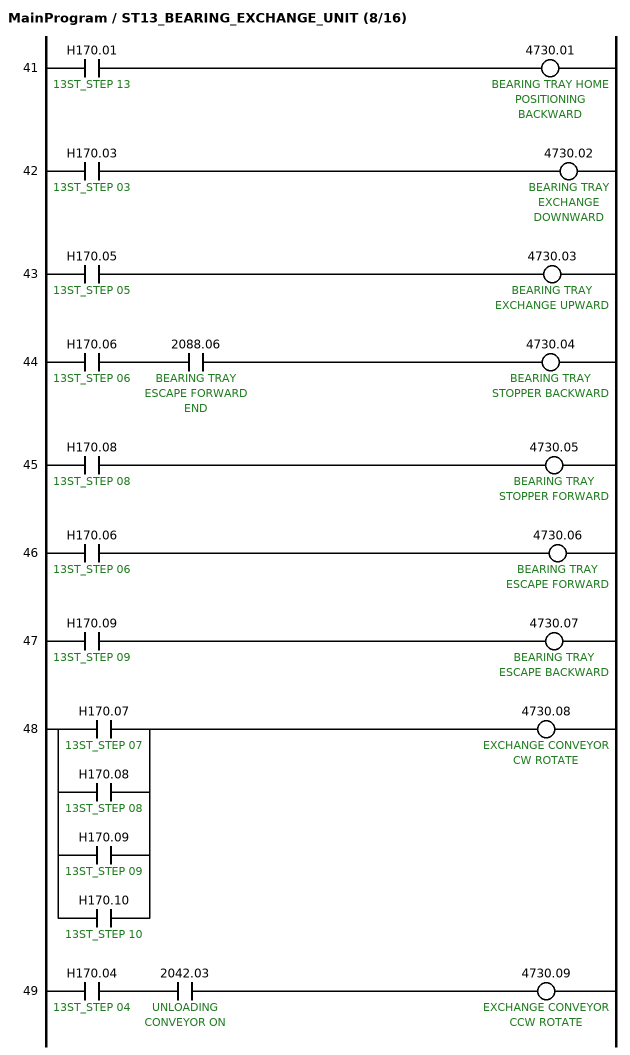
; [picture p600: MainProgram / ST13_BEARING_EXCHANGE_UNIT, rungs 41-49]
; rung 41
LD H170.01  ; 13ST_STEP 13
OUT 4730.01  ; BEARING TRAY HOME POSITIONING BACKWARD
; rung 42
LD H170.03  ; 13ST_STEP 03
OUT 4730.02  ; BEARING TRAY EXCHANGE DOWNWARD
; rung 43
LD H170.05  ; 13ST_STEP 05
OUT 4730.03  ; BEARING TRAY EXCHANGE UPWARD
; rung 44
LD H170.06  ; 13ST_STEP 06
AND 2088.06  ; BEARING TRAY ESCAPE FORWARD END
OUT 4730.04  ; BEARING TRAY STOPPER BACKWARD
; rung 45
LD H170.08  ; 13ST_STEP 08
OUT 4730.05  ; BEARING TRAY STOPPER FORWARD
; rung 46
LD H170.06  ; 13ST_STEP 06
OUT 4730.06  ; BEARING TRAY ESCAPE FORWARD
; rung 47
LD H170.09  ; 13ST_STEP 09
OUT 4730.07  ; BEARING TRAY ESCAPE BACKWARD
; rung 48
LD H170.07  ; 13ST_STEP 07
OR H170.08  ; 13ST_STEP 08
OR H170.09  ; 13ST_STEP 09
OR H170.10  ; 13ST_STEP 10
OUT 4730.08  ; EXCHANGE CONVEYOR CW ROTATE
; rung 49
LD H170.04  ; 13ST_STEP 04
AND 2042.03  ; UNLOADING CONVEYOR ON
OUT 4730.09  ; EXCHANGE CONVEYOR CCW ROTATE

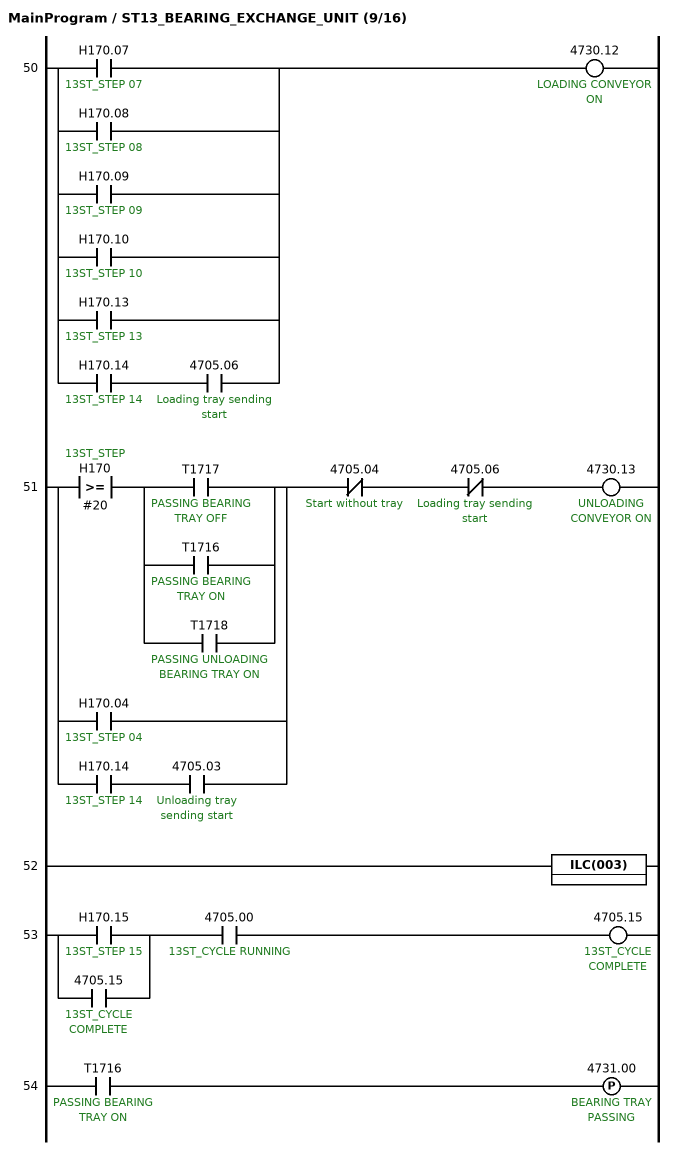
; rung 50
LD H170.07  ; 13ST_STEP 07
OR H170.08  ; 13ST_STEP 08
OR H170.09  ; 13ST_STEP 09
OR H170.10  ; 13ST_STEP 10
OR H170.13  ; 13ST_STEP 13
LD H170.14  ; 13ST_STEP 14
AND 4705.06  ; Loading tray sending start
ORLD
OUT 4730.12  ; LOADING CONVEYOR ON
; rung 51
LD>=(325) H170 #20  ; 13ST_STEP
LD T1717  ; PASSING BEARING TRAY OFF
OR T1716  ; PASSING BEARING TRAY ON
OR T1718  ; PASSING UNLOADING BEARING TRAY ON
ANDLD
OR H170.04  ; 13ST_STEP 04
LD H170.14  ; 13ST_STEP 14
AND 4705.03  ; Unloading tray sending start
ORLD
ANDNOT 4705.04  ; Start without tray
ANDNOT 4705.06  ; Loading tray sending start
OUT 4730.13  ; UNLOADING CONVEYOR ON
; rung 52
ILC(003)
; rung 53
LD H170.15  ; 13ST_STEP 15
OR 4705.15  ; 13ST_CYCLE COMPLETE
AND 4705.00  ; 13ST_CYCLE RUNNING
OUT 4705.15  ; 13ST_CYCLE COMPLETE
; rung 54
LD T1716  ; PASSING BEARING TRAY ON
DIFU(013) 4731.00  ; BEARING TRAY PASSING

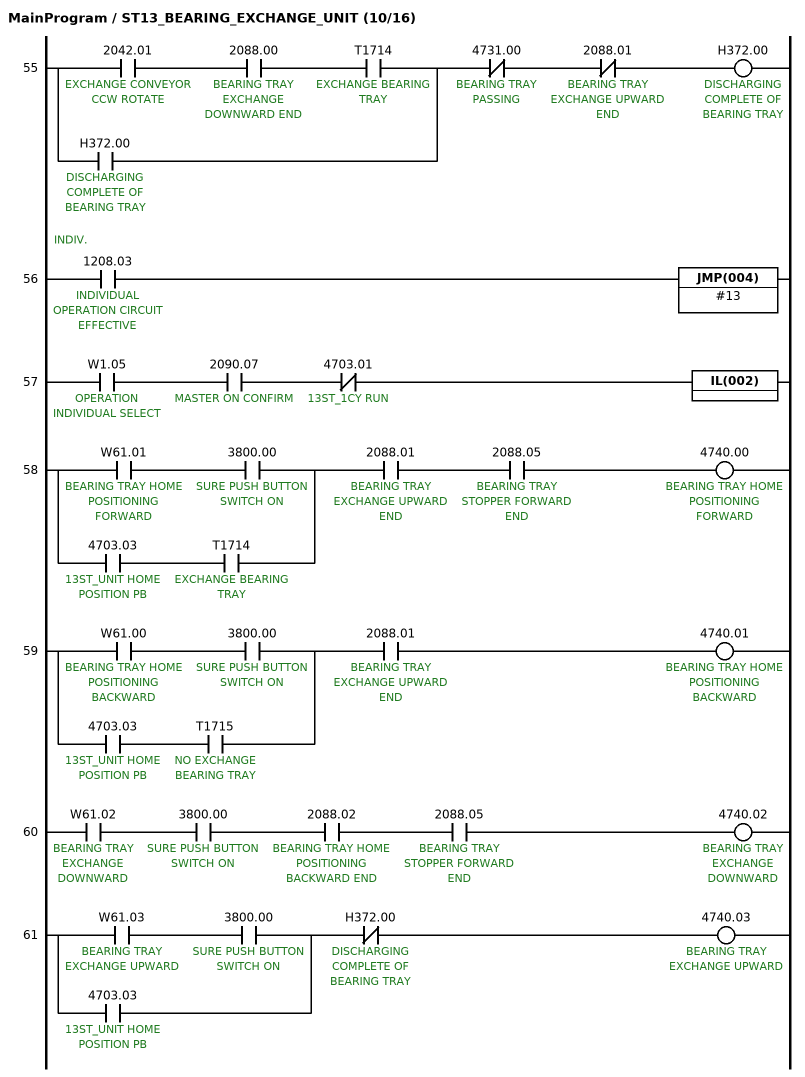
; rung 55
LD 2042.01  ; EXCHANGE CONVEYOR CCW ROTATE
AND 2088.00  ; BEARING TRAY EXCHANGE DOWNWARD END
AND T1714  ; EXCHANGE BEARING TRAY
OR H372.00  ; DISCHARGING COMPLETE OF BEARING TRAY
ANDNOT 4731.00  ; BEARING TRAY PASSING
ANDNOT 2088.01  ; BEARING TRAY EXCHANGE UPWARD END
OUT H372.00  ; DISCHARGING COMPLETE OF BEARING TRAY
; rung 56: INDIV.
LD 1208.03  ; INDIVIDUAL OPERATION CIRCUIT EFFECTIVE
JMP(004) #13
; rung 57
LD W1.05  ; OPERATION INDIVIDUAL SELECT
AND 2090.07  ; MASTER ON CONFIRM
ANDNOT 4703.01  ; 13ST_1CY RUN
IL(002)
; rung 58
LD W61.01  ; BEARING TRAY HOME POSITIONING FORWARD
AND 3800.00  ; SURE PUSH BUTTON SWITCH ON
LD 4703.03  ; 13ST_UNIT HOME POSITION PB
AND T1714  ; EXCHANGE BEARING TRAY
ORLD
AND 2088.01  ; BEARING TRAY EXCHANGE UPWARD END
AND 2088.05  ; BEARING TRAY STOPPER FORWARD END
OUT 4740.00  ; BEARING TRAY HOME POSITIONING FORWARD
; rung 59
LD W61.00  ; BEARING TRAY HOME POSITIONING BACKWARD
AND 3800.00  ; SURE PUSH BUTTON SWITCH ON
LD 4703.03  ; 13ST_UNIT HOME POSITION PB
AND T1715  ; NO EXCHANGE BEARING TRAY
ORLD
AND 2088.01  ; BEARING TRAY EXCHANGE UPWARD END
OUT 4740.01  ; BEARING TRAY HOME POSITIONING BACKWARD
; rung 60
LD W61.02  ; BEARING TRAY EXCHANGE DOWNWARD
AND 3800.00  ; SURE PUSH BUTTON SWITCH ON
AND 2088.02  ; BEARING TRAY HOME POSITIONING BACKWARD END
AND 2088.05  ; BEARING TRAY STOPPER FORWARD END
OUT 4740.02  ; BEARING TRAY EXCHANGE DOWNWARD
; rung 61
LD W61.03  ; BEARING TRAY EXCHANGE UPWARD
AND 3800.00  ; SURE PUSH BUTTON SWITCH ON
OR 4703.03  ; 13ST_UNIT HOME POSITION PB
ANDNOT H372.00  ; DISCHARGING COMPLETE OF BEARING TRAY
OUT 4740.03  ; BEARING TRAY EXCHANGE UPWARD

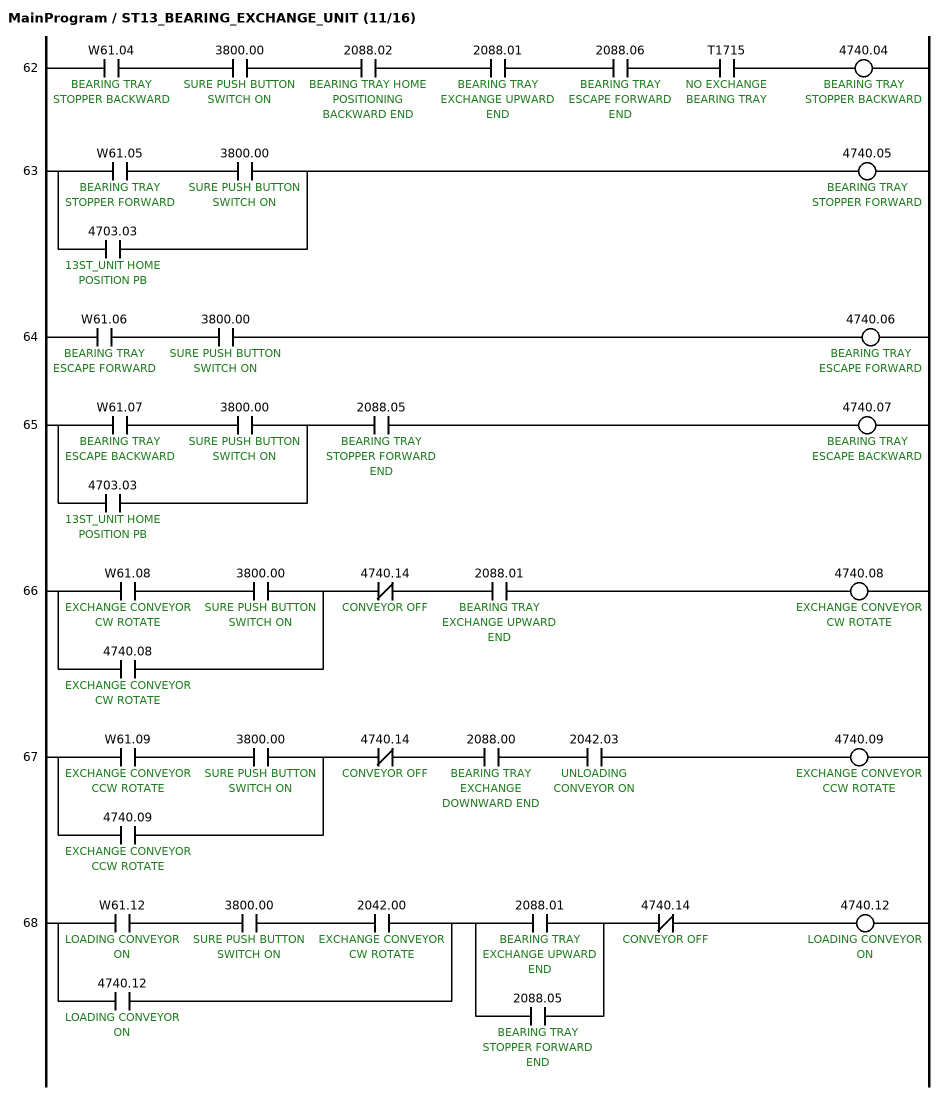
; rung 62
LD W61.04  ; BEARING TRAY STOPPER BACKWARD
AND 3800.00  ; SURE PUSH BUTTON SWITCH ON
AND 2088.02  ; BEARING TRAY HOME POSITIONING BACKWARD END
AND 2088.01  ; BEARING TRAY EXCHANGE UPWARD END
AND 2088.06  ; BEARING TRAY ESCAPE FORWARD END
AND T1715  ; NO EXCHANGE BEARING TRAY
OUT 4740.04  ; BEARING TRAY STOPPER BACKWARD
; rung 63
LD W61.05  ; BEARING TRAY STOPPER FORWARD
AND 3800.00  ; SURE PUSH BUTTON SWITCH ON
OR 4703.03  ; 13ST_UNIT HOME POSITION PB
OUT 4740.05  ; BEARING TRAY STOPPER FORWARD
; rung 64
LD W61.06  ; BEARING TRAY ESCAPE FORWARD
AND 3800.00  ; SURE PUSH BUTTON SWITCH ON
OUT 4740.06  ; BEARING TRAY ESCAPE FORWARD
; rung 65
LD W61.07  ; BEARING TRAY ESCAPE BACKWARD
AND 3800.00  ; SURE PUSH BUTTON SWITCH ON
OR 4703.03  ; 13ST_UNIT HOME POSITION PB
AND 2088.05  ; BEARING TRAY STOPPER FORWARD END
OUT 4740.07  ; BEARING TRAY ESCAPE BACKWARD
; rung 66
LD W61.08  ; EXCHANGE CONVEYOR CW ROTATE
AND 3800.00  ; SURE PUSH BUTTON SWITCH ON
OR 4740.08  ; EXCHANGE CONVEYOR CW ROTATE
ANDNOT 4740.14  ; CONVEYOR OFF
AND 2088.01  ; BEARING TRAY EXCHANGE UPWARD END
OUT 4740.08  ; EXCHANGE CONVEYOR CW ROTATE
; rung 67
LD W61.09  ; EXCHANGE CONVEYOR CCW ROTATE
AND 3800.00  ; SURE PUSH BUTTON SWITCH ON
OR 4740.09  ; EXCHANGE CONVEYOR CCW ROTATE
ANDNOT 4740.14  ; CONVEYOR OFF
AND 2088.00  ; BEARING TRAY EXCHANGE DOWNWARD END
AND 2042.03  ; UNLOADING CONVEYOR ON
OUT 4740.09  ; EXCHANGE CONVEYOR CCW ROTATE
; rung 68
LD W61.12  ; LOADING CONVEYOR ON
AND 3800.00  ; SURE PUSH BUTTON SWITCH ON
AND 2042.00  ; EXCHANGE CONVEYOR CW ROTATE
OR 4740.12  ; LOADING CONVEYOR ON
LD 2088.01  ; BEARING TRAY EXCHANGE UPWARD END
OR 2088.05  ; BEARING TRAY STOPPER FORWARD END
ANDLD
ANDNOT 4740.14  ; CONVEYOR OFF
OUT 4740.12  ; LOADING CONVEYOR ON

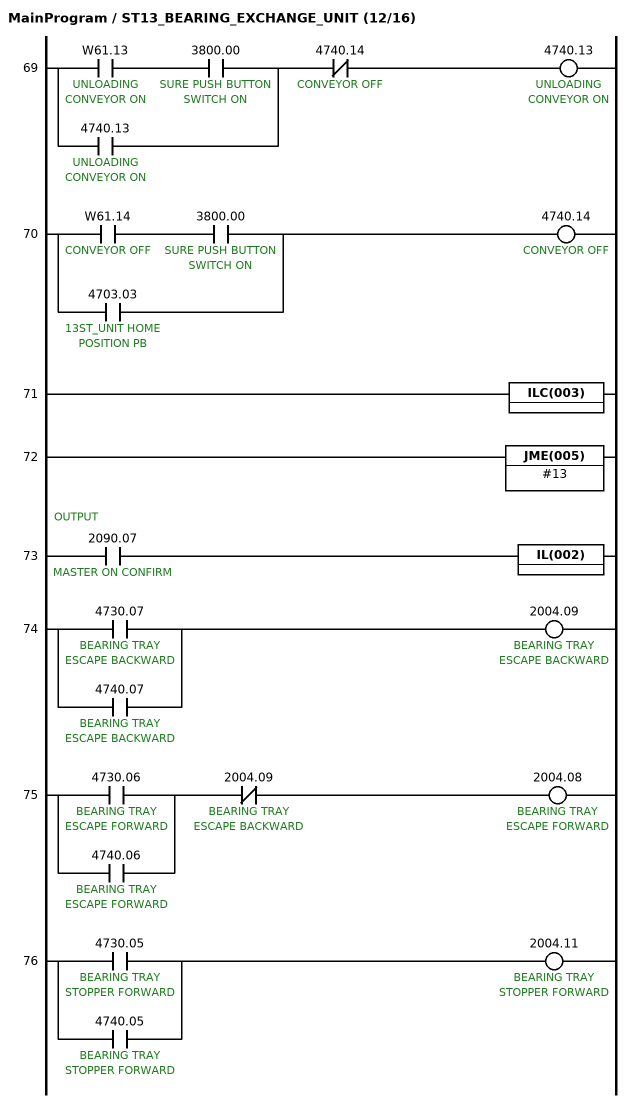
; rung 69
LD W61.13  ; UNLOADING CONVEYOR ON
AND 3800.00  ; SURE PUSH BUTTON SWITCH ON
OR 4740.13  ; UNLOADING CONVEYOR ON
ANDNOT 4740.14  ; CONVEYOR OFF
OUT 4740.13  ; UNLOADING CONVEYOR ON
; rung 70
LD W61.14  ; CONVEYOR OFF
AND 3800.00  ; SURE PUSH BUTTON SWITCH ON
OR 4703.03  ; 13ST_UNIT HOME POSITION PB
OUT 4740.14  ; CONVEYOR OFF
; rung 71
ILC(003)
; rung 72
JME(005) #13
; rung 73: OUTPUT
LD 2090.07  ; MASTER ON CONFIRM
IL(002)
; rung 74
LD 4730.07  ; BEARING TRAY ESCAPE BACKWARD
OR 4740.07  ; BEARING TRAY ESCAPE BACKWARD
OUT 2004.09  ; BEARING TRAY ESCAPE BACKWARD
; rung 75
LD 4730.06  ; BEARING TRAY ESCAPE FORWARD
OR 4740.06  ; BEARING TRAY ESCAPE FORWARD
ANDNOT 2004.09  ; BEARING TRAY ESCAPE BACKWARD
OUT 2004.08  ; BEARING TRAY ESCAPE FORWARD
; rung 76
LD 4730.05  ; BEARING TRAY STOPPER FORWARD
OR 4740.05  ; BEARING TRAY STOPPER FORWARD
OUT 2004.11  ; BEARING TRAY STOPPER FORWARD

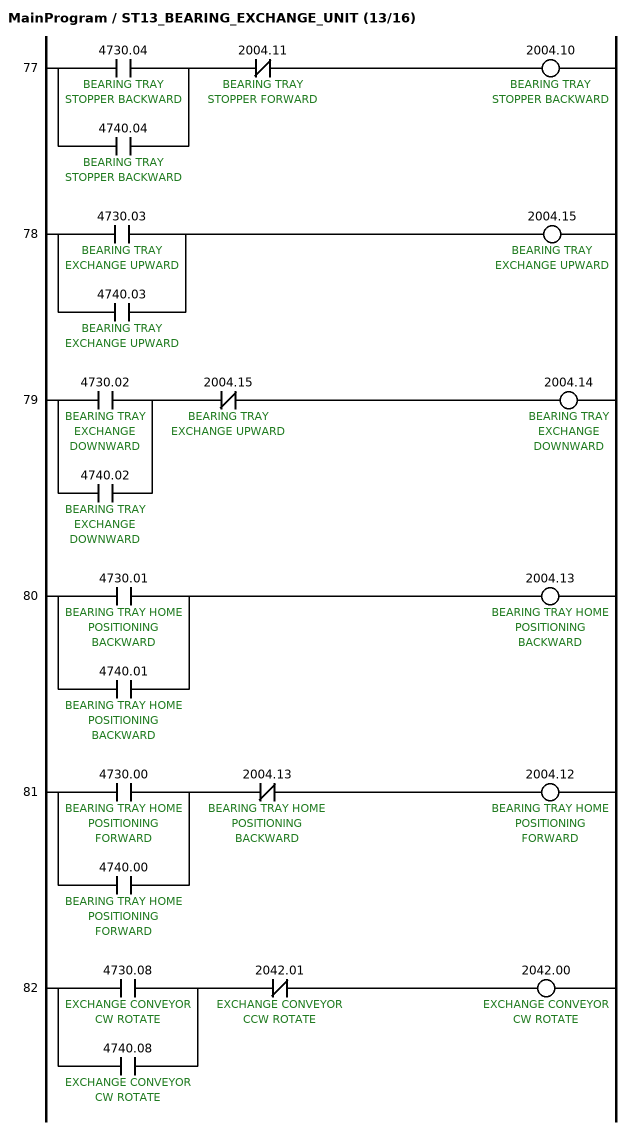
; rung 77
LD 4730.04  ; BEARING TRAY STOPPER BACKWARD
OR 4740.04  ; BEARING TRAY STOPPER BACKWARD
ANDNOT 2004.11  ; BEARING TRAY STOPPER FORWARD
OUT 2004.10  ; BEARING TRAY STOPPER BACKWARD
; rung 78
LD 4730.03  ; BEARING TRAY EXCHANGE UPWARD
OR 4740.03  ; BEARING TRAY EXCHANGE UPWARD
OUT 2004.15  ; BEARING TRAY EXCHANGE UPWARD
; rung 79
LD 4730.02  ; BEARING TRAY EXCHANGE DOWNWARD
OR 4740.02  ; BEARING TRAY EXCHANGE DOWNWARD
ANDNOT 2004.15  ; BEARING TRAY EXCHANGE UPWARD
OUT 2004.14  ; BEARING TRAY EXCHANGE DOWNWARD
; rung 80
LD 4730.01  ; BEARING TRAY HOME POSITIONING BACKWARD
OR 4740.01  ; BEARING TRAY HOME POSITIONING BACKWARD
OUT 2004.13  ; BEARING TRAY HOME POSITIONING BACKWARD
; rung 81
LD 4730.00  ; BEARING TRAY HOME POSITIONING FORWARD
OR 4740.00  ; BEARING TRAY HOME POSITIONING FORWARD
ANDNOT 2004.13  ; BEARING TRAY HOME POSITIONING BACKWARD
OUT 2004.12  ; BEARING TRAY HOME POSITIONING FORWARD
; rung 82
LD 4730.08  ; EXCHANGE CONVEYOR CW ROTATE
OR 4740.08  ; EXCHANGE CONVEYOR CW ROTATE
ANDNOT 2042.01  ; EXCHANGE CONVEYOR CCW ROTATE
OUT 2042.00  ; EXCHANGE CONVEYOR CW ROTATE

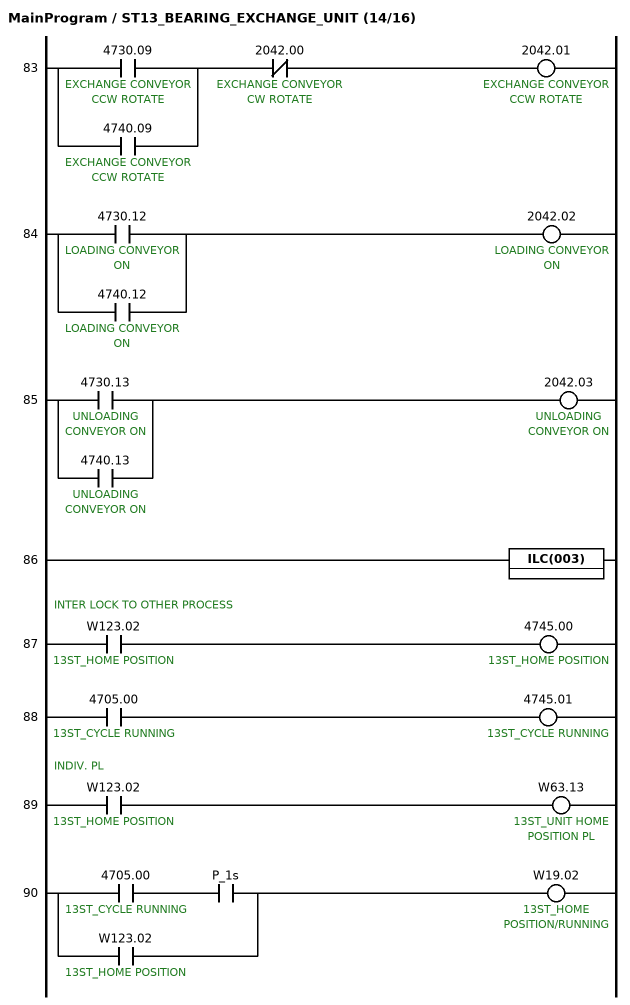
; rung 83
LD 4730.09  ; EXCHANGE CONVEYOR CCW ROTATE
OR 4740.09  ; EXCHANGE CONVEYOR CCW ROTATE
ANDNOT 2042.00  ; EXCHANGE CONVEYOR CW ROTATE
OUT 2042.01  ; EXCHANGE CONVEYOR CCW ROTATE
; rung 84
LD 4730.12  ; LOADING CONVEYOR ON
OR 4740.12  ; LOADING CONVEYOR ON
OUT 2042.02  ; LOADING CONVEYOR ON
; rung 85
LD 4730.13  ; UNLOADING CONVEYOR ON
OR 4740.13  ; UNLOADING CONVEYOR ON
OUT 2042.03  ; UNLOADING CONVEYOR ON
; rung 86
ILC(003)
; rung 87: INTER LOCK TO OTHER PROCESS
LD W123.02  ; 13ST_HOME POSITION
OUT 4745.00  ; 13ST_HOME POSITION
; rung 88
LD 4705.00  ; 13ST_CYCLE RUNNING
OUT 4745.01  ; 13ST_CYCLE RUNNING
; rung 89: INDIV. PL
LD W123.02  ; 13ST_HOME POSITION
OUT W63.13  ; 13ST_UNIT HOME POSITION PL
; rung 90
LD 4705.00  ; 13ST_CYCLE RUNNING
AND P_1s
OR W123.02  ; 13ST_HOME POSITION
OUT W19.02  ; 13ST_HOME POSITION/RUNNING

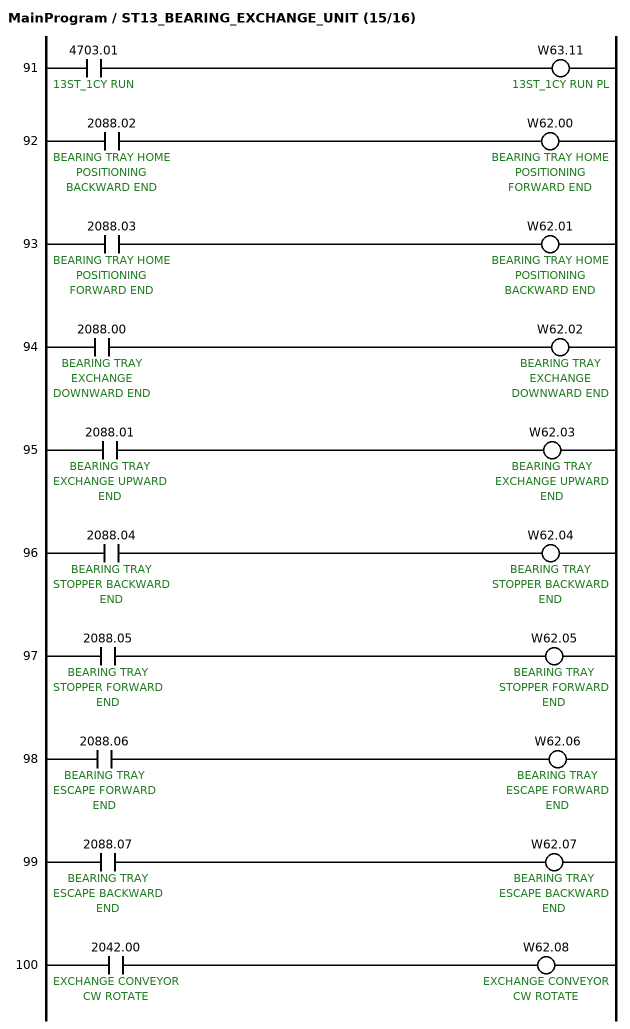
; rung 91
LD 4703.01  ; 13ST_1CY RUN
OUT W63.11  ; 13ST_1CY RUN PL
; rung 92
LD 2088.02  ; BEARING TRAY HOME POSITIONING BACKWARD END
OUT W62.00  ; BEARING TRAY HOME POSITIONING FORWARD END
; rung 93
LD 2088.03  ; BEARING TRAY HOME POSITIONING FORWARD END
OUT W62.01  ; BEARING TRAY HOME POSITIONING BACKWARD END
; rung 94
LD 2088.00  ; BEARING TRAY EXCHANGE DOWNWARD END
OUT W62.02  ; BEARING TRAY EXCHANGE DOWNWARD END
; rung 95
LD 2088.01  ; BEARING TRAY EXCHANGE UPWARD END
OUT W62.03  ; BEARING TRAY EXCHANGE UPWARD END
; rung 96
LD 2088.04  ; BEARING TRAY STOPPER BACKWARD END
OUT W62.04  ; BEARING TRAY STOPPER BACKWARD END
; rung 97
LD 2088.05  ; BEARING TRAY STOPPER FORWARD END
OUT W62.05  ; BEARING TRAY STOPPER FORWARD END
; rung 98
LD 2088.06  ; BEARING TRAY ESCAPE FORWARD END
OUT W62.06  ; BEARING TRAY ESCAPE FORWARD END
; rung 99
LD 2088.07  ; BEARING TRAY ESCAPE BACKWARD END
OUT W62.07  ; BEARING TRAY ESCAPE BACKWARD END
; rung 100
LD 2042.00  ; EXCHANGE CONVEYOR CW ROTATE
OUT W62.08  ; EXCHANGE CONVEYOR CW ROTATE

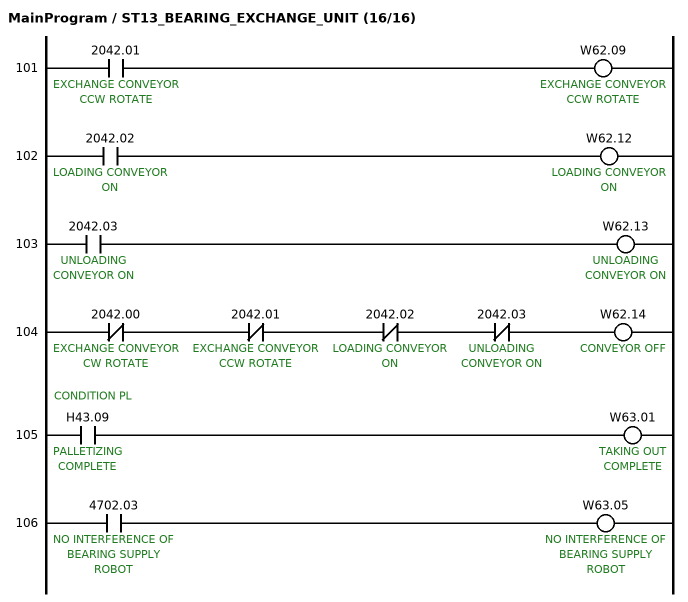
; rung 101
LD 2042.01  ; EXCHANGE CONVEYOR CCW ROTATE
OUT W62.09  ; EXCHANGE CONVEYOR CCW ROTATE
; rung 102
LD 2042.02  ; LOADING CONVEYOR ON
OUT W62.12  ; LOADING CONVEYOR ON
; rung 103
LD 2042.03  ; UNLOADING CONVEYOR ON
OUT W62.13  ; UNLOADING CONVEYOR ON
; rung 104
LDNOT 2042.00  ; EXCHANGE CONVEYOR CW ROTATE
ANDNOT 2042.01  ; EXCHANGE CONVEYOR CCW ROTATE
ANDNOT 2042.02  ; LOADING CONVEYOR ON
ANDNOT 2042.03  ; UNLOADING CONVEYOR ON
OUT W62.14  ; CONVEYOR OFF
; rung 105: CONDITION PL
LD H43.09  ; PALLETIZING COMPLETE
OUT W63.01  ; TAKING OUT COMPLETE
; rung 106
LD 4702.03  ; NO INTERFERENCE OF BEARING SUPPLY ROBOT
OUT W63.05  ; NO INTERFERENCE OF BEARING SUPPLY ROBOT

### Section ST14_DEFECT_DISCHARGE_UNIT
; rung 0: 14ST_DEFECT DISCHARGE UNIT

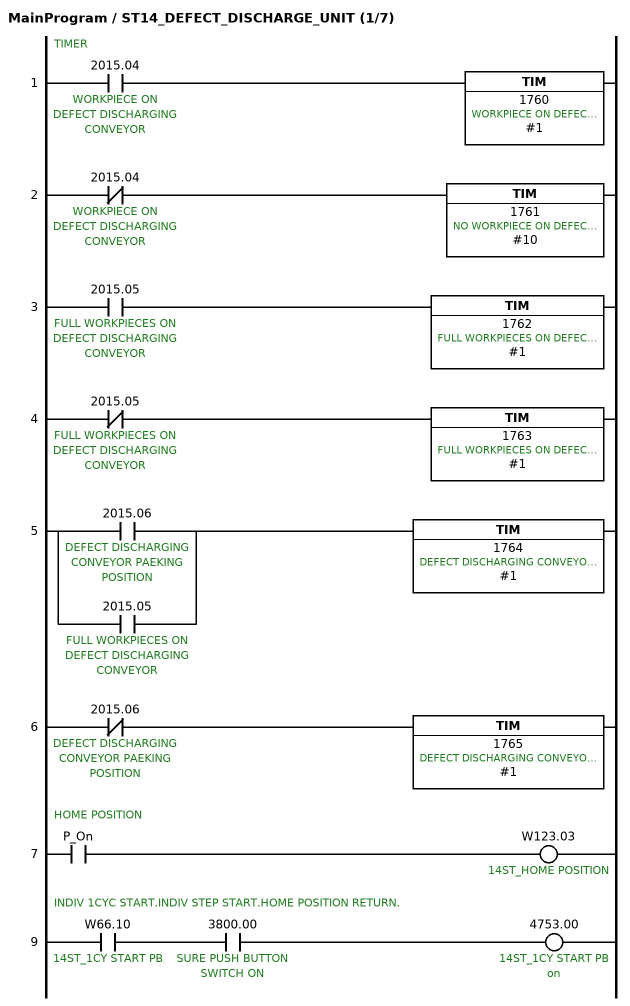
; rung 1: TIMER
LD 2015.04  ; WORKPIECE ON DEFECT DISCHARGING CONVEYOR
TIM 1760 #1  ; WORKPIECE ON DEFECT DISCHARGING CONVEYOR
; rung 2
LDNOT 2015.04  ; WORKPIECE ON DEFECT DISCHARGING CONVEYOR
TIM 1761 #10  ; NO WORKPIECE ON DEFECT DISCHARGING CONVEYOR
; rung 3
LD 2015.05  ; FULL WORKPIECES ON DEFECT DISCHARGING CONVEYOR
TIM 1762 #1  ; FULL WORKPIECES ON DEFECT DISCHARGING CONVEYOR IS TURNED ON
; rung 4
LDNOT 2015.05  ; FULL WORKPIECES ON DEFECT DISCHARGING CONVEYOR
TIM 1763 #1  ; FULL WORKPIECES ON DEFECT DISCHARGING CONVEYOR IS TURNED OFF
; rung 5
LD 2015.06  ; DEFECT DISCHARGING CONVEYOR PAEKING POSITION
OR 2015.05  ; FULL WORKPIECES ON DEFECT DISCHARGING CONVEYOR
TIM 1764 #1  ; DEFECT DISCHARGING CONVEYOR PAEKING POSITION IS TURNED ON
; rung 6
LDNOT 2015.06  ; DEFECT DISCHARGING CONVEYOR PAEKING POSITION
TIM 1765 #1  ; DEFECT DISCHARGING CONVEYOR PAEKING POSITION IS TURNED OFF
; rung 7: HOME POSITION
LD P_On
OUT W123.03  ; 14ST_HOME POSITION
; rung 8: INTERFERENCE
; rung 9: INDIV 1CYC START.INDIV STEP START.HOME POSITION RETURN.
LD W66.10  ; 14ST_1CY START PB
AND 3800.00  ; SURE PUSH BUTTON SWITCH ON
OUT 4753.00  ; 14ST_1CY START PB on

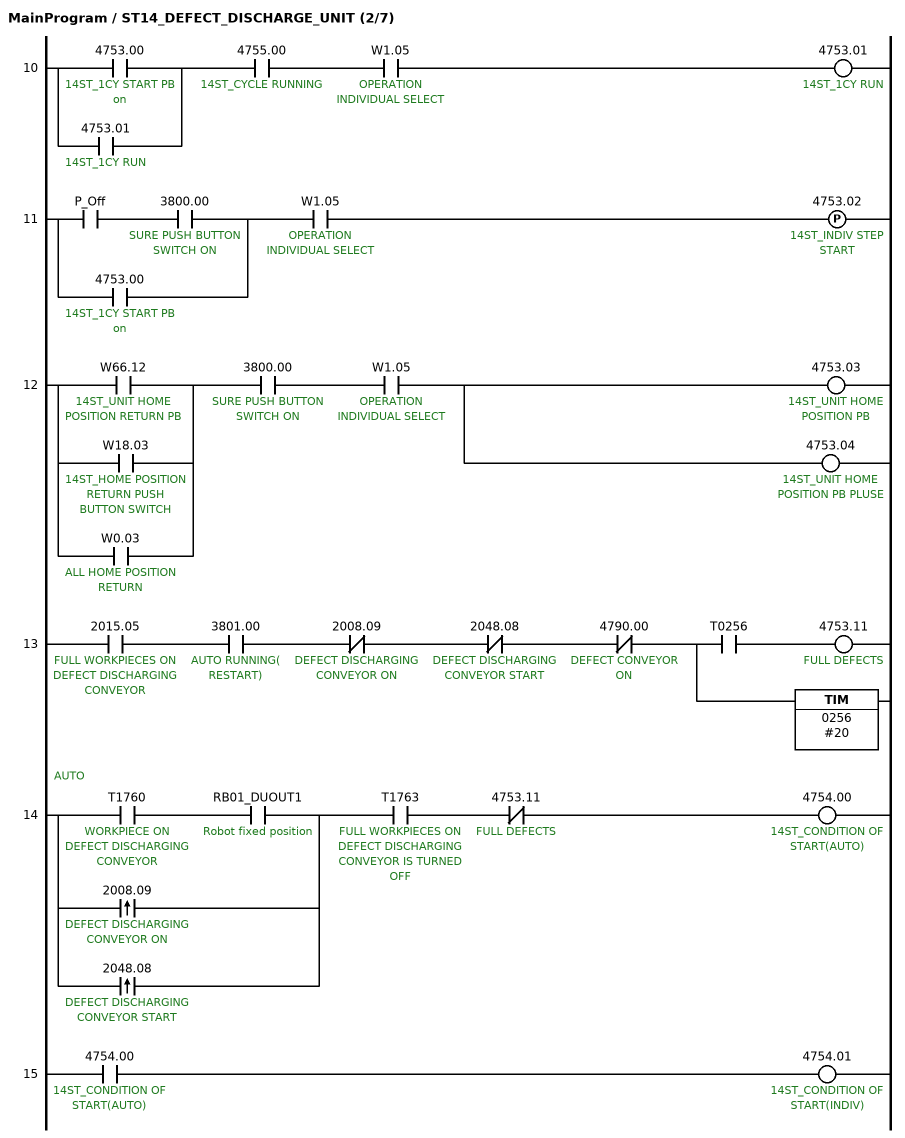
; rung 10
LD 4753.00  ; 14ST_1CY START PB on
OR 4753.01  ; 14ST_1CY RUN
AND 4755.00  ; 14ST_CYCLE RUNNING
AND W1.05  ; OPERATION INDIVIDUAL SELECT
OUT 4753.01  ; 14ST_1CY RUN
; rung 11
LD P_Off
AND 3800.00  ; SURE PUSH BUTTON SWITCH ON
OR 4753.00  ; 14ST_1CY START PB on
AND W1.05  ; OPERATION INDIVIDUAL SELECT
DIFU(013) 4753.02  ; 14ST_INDIV STEP START
; rung 12
LD W66.12  ; 14ST_UNIT HOME POSITION RETURN PB
OR W18.03  ; 14ST_HOME POSITION RETURN PUSH BUTTON SWITCH
OR W0.03  ; ALL HOME POSITION RETURN
AND 3800.00  ; SURE PUSH BUTTON SWITCH ON
AND W1.05  ; OPERATION INDIVIDUAL SELECT
OUT 4753.03  ; 14ST_UNIT HOME POSITION PB
OUT 4753.04  ; 14ST_UNIT HOME POSITION PB PLUSE
; rung 13
LD 2015.05  ; FULL WORKPIECES ON DEFECT DISCHARGING CONVEYOR
AND 3801.00  ; AUTO RUNNING(RESTART)
ANDNOT 2008.09  ; DEFECT DISCHARGING CONVEYOR ON
ANDNOT 2048.08  ; DEFECT DISCHARGING CONVEYOR START
ANDNOT 4790.00  ; DEFECT CONVEYOR ON
OUT TR0
AND T0256
OUT 4753.11  ; FULL DEFECTS
LD TR0
TIM 0256 #20
; rung 14: AUTO
LD T1760  ; WORKPIECE ON DEFECT DISCHARGING CONVEYOR
AND RB01_DUOUT1  ; Robot fixed position
@OR 2008.09  ; DEFECT DISCHARGING CONVEYOR ON
@OR 2048.08  ; DEFECT DISCHARGING CONVEYOR START
AND T1763  ; FULL WORKPIECES ON DEFECT DISCHARGING CONVEYOR IS TURNED OFF
ANDNOT 4753.11  ; FULL DEFECTS
OUT 4754.00  ; 14ST_CONDITION OF START(AUTO)
; rung 15
LD 4754.00  ; 14ST_CONDITION OF START(AUTO)
OUT 4754.01  ; 14ST_CONDITION OF START(INDIV)

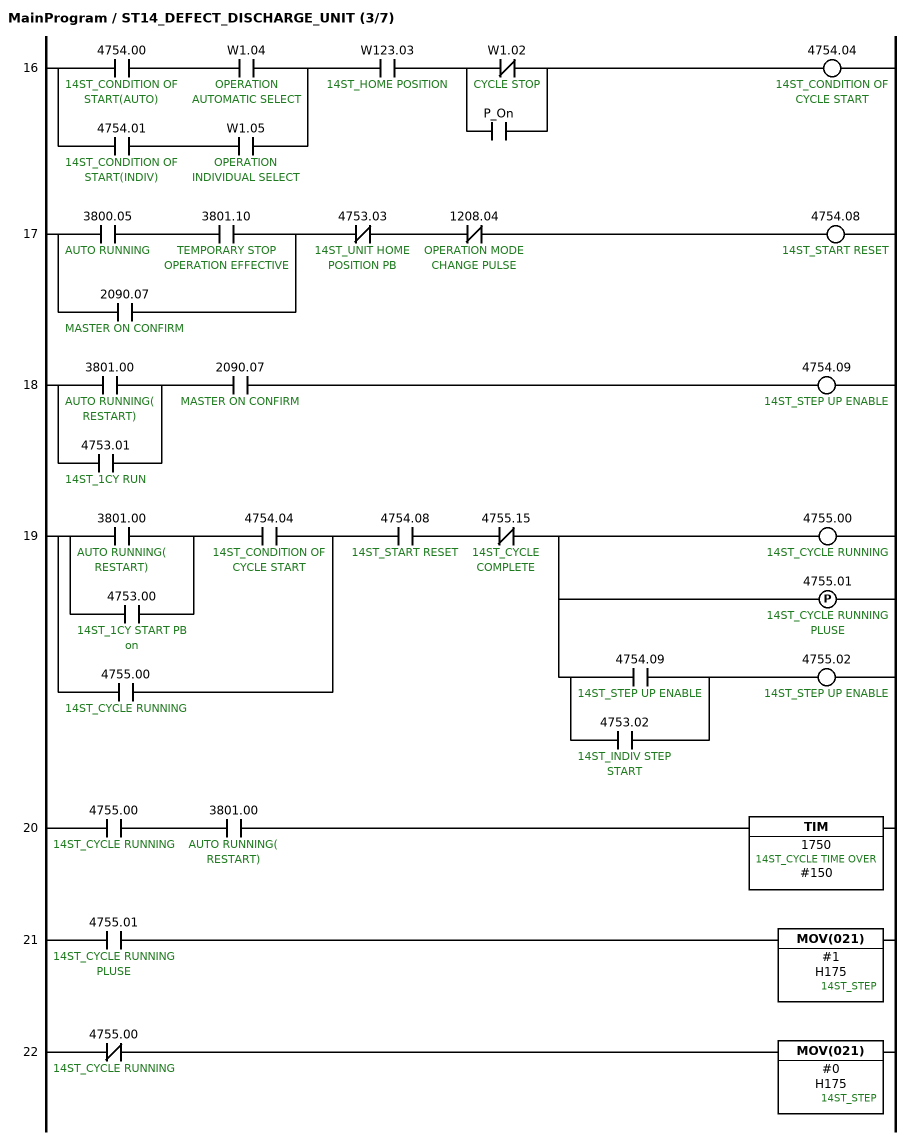
; rung 16
LD 4754.00  ; 14ST_CONDITION OF START(AUTO)
AND W1.04  ; OPERATION AUTOMATIC SELECT
LD 4754.01  ; 14ST_CONDITION OF START(INDIV)
AND W1.05  ; OPERATION INDIVIDUAL SELECT
ORLD
AND W123.03  ; 14ST_HOME POSITION
LDNOT W1.02  ; CYCLE STOP
OR P_On
ANDLD
OUT 4754.04  ; 14ST_CONDITION OF CYCLE START
; rung 17
LD 3800.05  ; AUTO RUNNING
AND 3801.10  ; TEMPORARY STOP OPERATION EFFECTIVE
OR 2090.07  ; MASTER ON CONFIRM
ANDNOT 4753.03  ; 14ST_UNIT HOME POSITION PB
ANDNOT 1208.04  ; OPERATION MODE CHANGE PULSE
OUT 4754.08  ; 14ST_START RESET
; rung 18
LD 3801.00  ; AUTO RUNNING(RESTART)
OR 4753.01  ; 14ST_1CY RUN
AND 2090.07  ; MASTER ON CONFIRM
OUT 4754.09  ; 14ST_STEP UP ENABLE
; rung 19
LD 3801.00  ; AUTO RUNNING(RESTART)
OR 4753.00  ; 14ST_1CY START PB on
AND 4754.04  ; 14ST_CONDITION OF CYCLE START
OR 4755.00  ; 14ST_CYCLE RUNNING
AND 4754.08  ; 14ST_START RESET
ANDNOT 4755.15  ; 14ST_CYCLE COMPLETE
OUT 4755.00  ; 14ST_CYCLE RUNNING
DIFU(013) 4755.01  ; 14ST_CYCLE RUNNING PLUSE
LD 4754.09  ; 14ST_STEP UP ENABLE
OR 4753.02  ; 14ST_INDIV STEP START
ANDLD
OUT 4755.02  ; 14ST_STEP UP ENABLE
; rung 20
LD 4755.00  ; 14ST_CYCLE RUNNING
AND 3801.00  ; AUTO RUNNING(RESTART)
TIM 1750 #150  ; 14ST_CYCLE TIME OVER
; rung 21
LD 4755.01  ; 14ST_CYCLE RUNNING PLUSE
MOV(021) #1 H175  ; 14ST_STEP
; rung 22
LDNOT 4755.00  ; 14ST_CYCLE RUNNING
MOV(021) #0 H175  ; 14ST_STEP

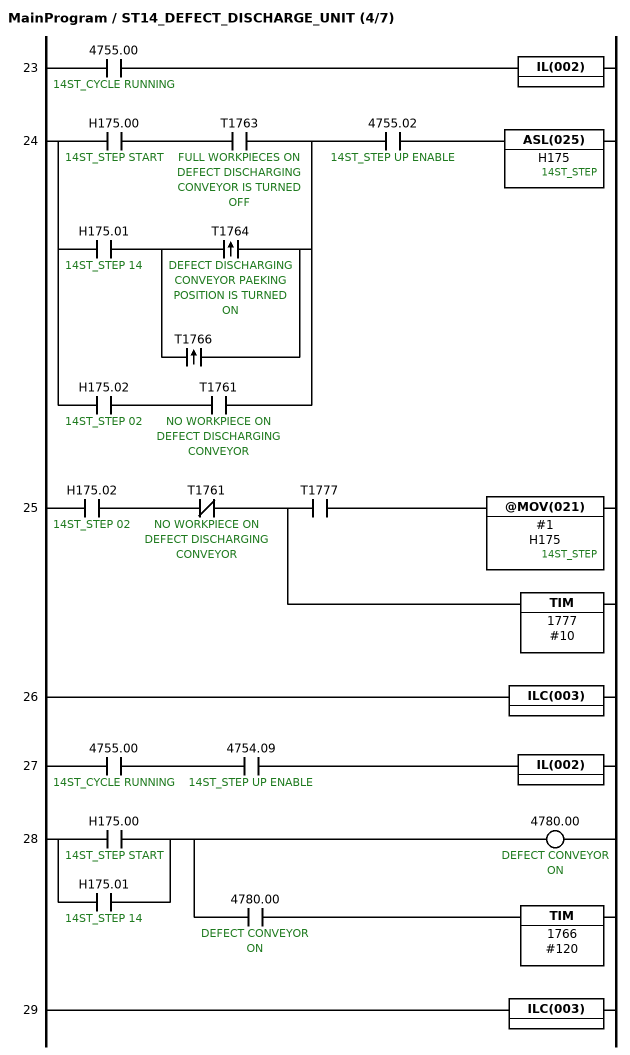
; rung 23
LD 4755.00  ; 14ST_CYCLE RUNNING
IL(002)
; rung 24
LD H175.00  ; 14ST_STEP START
AND T1763  ; FULL WORKPIECES ON DEFECT DISCHARGING CONVEYOR IS TURNED OFF
LD H175.01  ; 14ST_STEP 14
@LD T1764  ; DEFECT DISCHARGING CONVEYOR PAEKING POSITION IS TURNED ON
@OR T1766
ANDLD
ORLD
LD H175.02  ; 14ST_STEP 02
AND T1761  ; NO WORKPIECE ON DEFECT DISCHARGING CONVEYOR
ORLD
AND 4755.02  ; 14ST_STEP UP ENABLE
ASL(025) H175  ; 14ST_STEP
; rung 25
LD H175.02  ; 14ST_STEP 02
ANDNOT T1761  ; NO WORKPIECE ON DEFECT DISCHARGING CONVEYOR
OUT TR0
AND T1777
@MOV(021) #1 H175  ; 14ST_STEP
LD TR0
TIM 1777 #10
; rung 26
ILC(003)
; rung 27
LD 4755.00  ; 14ST_CYCLE RUNNING
AND 4754.09  ; 14ST_STEP UP ENABLE
IL(002)
; rung 28
LD H175.00  ; 14ST_STEP START
OR H175.01  ; 14ST_STEP 14
OUT 4780.00  ; DEFECT CONVEYOR ON
AND 4780.00  ; DEFECT CONVEYOR ON
TIM 1766 #120
; rung 29
ILC(003)

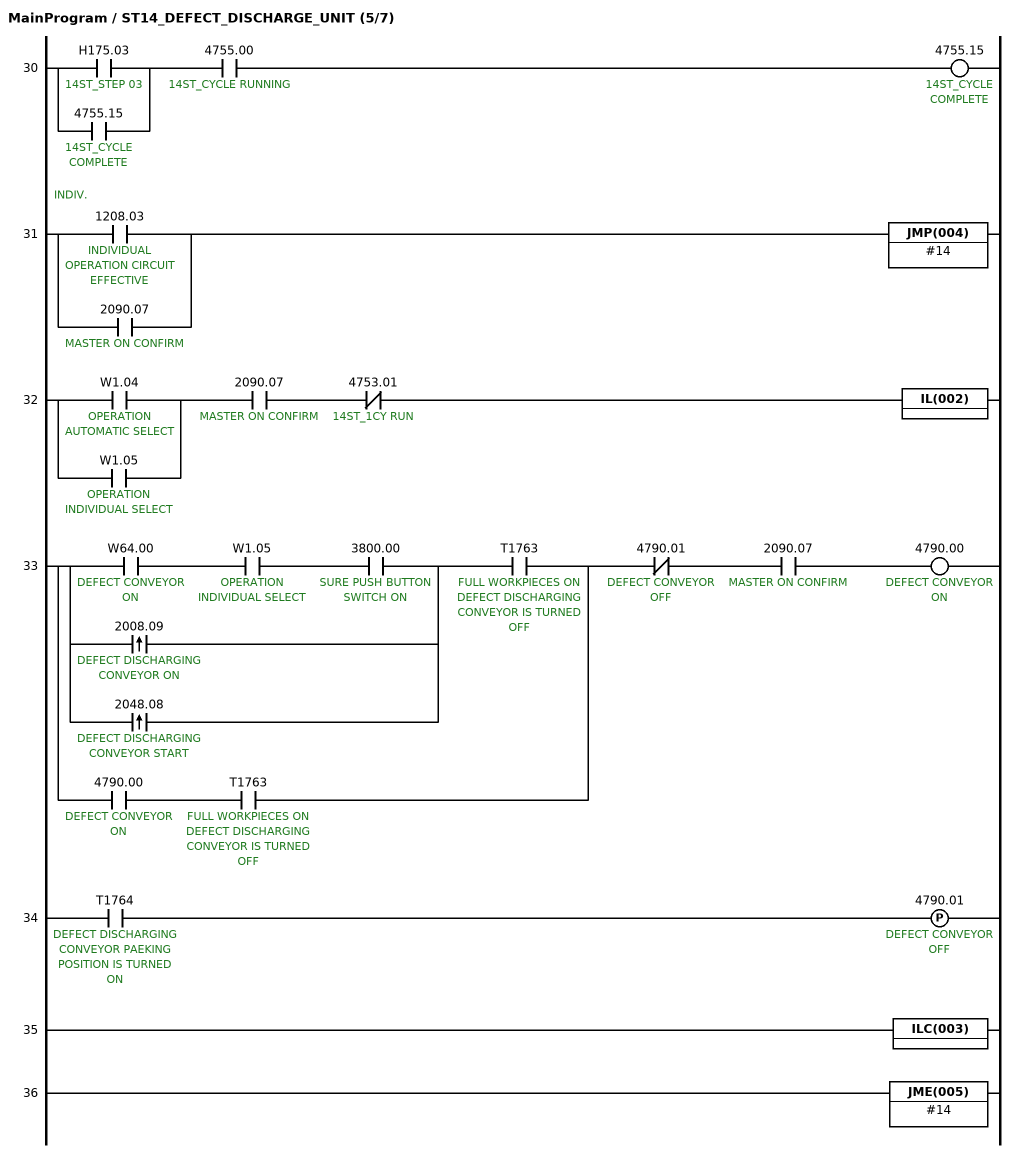
; rung 30
LD H175.03  ; 14ST_STEP 03
OR 4755.15  ; 14ST_CYCLE COMPLETE
AND 4755.00  ; 14ST_CYCLE RUNNING
OUT 4755.15  ; 14ST_CYCLE COMPLETE
; rung 31: INDIV.
LD 1208.03  ; INDIVIDUAL OPERATION CIRCUIT EFFECTIVE
OR 2090.07  ; MASTER ON CONFIRM
JMP(004) #14
; rung 32
LD W1.04  ; OPERATION AUTOMATIC SELECT
OR W1.05  ; OPERATION INDIVIDUAL SELECT
AND 2090.07  ; MASTER ON CONFIRM
ANDNOT 4753.01  ; 14ST_1CY RUN
IL(002)
; rung 33
LD W64.00  ; DEFECT CONVEYOR ON
AND W1.05  ; OPERATION INDIVIDUAL SELECT
AND 3800.00  ; SURE PUSH BUTTON SWITCH ON
@OR 2008.09  ; DEFECT DISCHARGING CONVEYOR ON
@OR 2048.08  ; DEFECT DISCHARGING CONVEYOR START
AND T1763  ; FULL WORKPIECES ON DEFECT DISCHARGING CONVEYOR IS TURNED OFF
LD 4790.00  ; DEFECT CONVEYOR ON
AND T1763  ; FULL WORKPIECES ON DEFECT DISCHARGING CONVEYOR IS TURNED OFF
ORLD
ANDNOT 4790.01  ; DEFECT CONVEYOR OFF
AND 2090.07  ; MASTER ON CONFIRM
OUT 4790.00  ; DEFECT CONVEYOR ON
; rung 34
LD T1764  ; DEFECT DISCHARGING CONVEYOR PAEKING POSITION IS TURNED ON
DIFU(013) 4790.01  ; DEFECT CONVEYOR OFF
; rung 35
ILC(003)
; rung 36
JME(005) #14

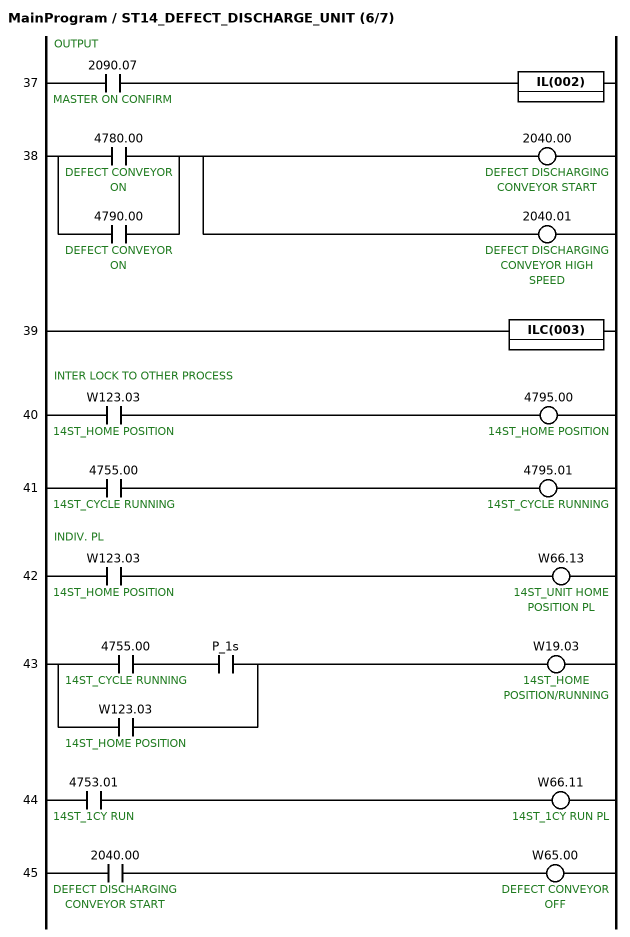
; rung 37: OUTPUT
LD 2090.07  ; MASTER ON CONFIRM
IL(002)
; rung 38
LD 4780.00  ; DEFECT CONVEYOR ON
OR 4790.00  ; DEFECT CONVEYOR ON
OUT 2040.00  ; DEFECT DISCHARGING CONVEYOR START
OUT 2040.01  ; DEFECT DISCHARGING CONVEYOR HIGH SPEED
; rung 39
ILC(003)
; rung 40: INTER LOCK TO OTHER PROCESS
LD W123.03  ; 14ST_HOME POSITION
OUT 4795.00  ; 14ST_HOME POSITION
; rung 41
LD 4755.00  ; 14ST_CYCLE RUNNING
OUT 4795.01  ; 14ST_CYCLE RUNNING
; rung 42: INDIV. PL
LD W123.03  ; 14ST_HOME POSITION
OUT W66.13  ; 14ST_UNIT HOME POSITION PL
; rung 43
LD 4755.00  ; 14ST_CYCLE RUNNING
AND P_1s
OR W123.03  ; 14ST_HOME POSITION
OUT W19.03  ; 14ST_HOME POSITION/RUNNING
; rung 44
LD 4753.01  ; 14ST_1CY RUN
OUT W66.11  ; 14ST_1CY RUN PL
; rung 45
LD 2040.00  ; DEFECT DISCHARGING CONVEYOR START
OUT W65.00  ; DEFECT CONVEYOR OFF

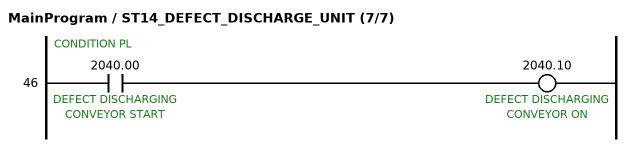
; rung 46: CONDITION PL
LD 2040.00  ; DEFECT DISCHARGING CONVEYOR START
OUT 2040.10  ; DEFECT DISCHARGING CONVEYOR ON

### Section ST15_LANE_1_PALLETIZING_UNIT

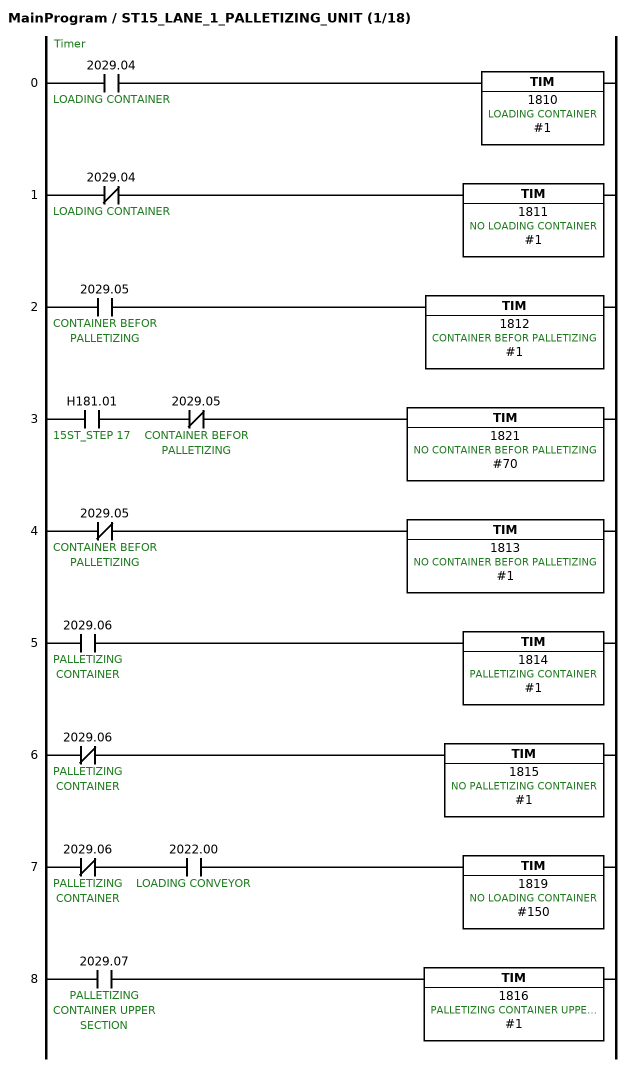
; rung 0: Timer
LD 2029.04  ; LOADING CONTAINER
TIM 1810 #1  ; LOADING CONTAINER
; rung 1
LDNOT 2029.04  ; LOADING CONTAINER
TIM 1811 #1  ; NO LOADING CONTAINER
; rung 2
LD 2029.05  ; CONTAINER BEFOR PALLETIZING
TIM 1812 #1  ; CONTAINER BEFOR PALLETIZING
; rung 3
LD H181.01  ; 15ST_STEP 17
ANDNOT 2029.05  ; CONTAINER BEFOR PALLETIZING
TIM 1821 #70  ; NO CONTAINER BEFOR PALLETIZING
; rung 4
LDNOT 2029.05  ; CONTAINER BEFOR PALLETIZING
TIM 1813 #1  ; NO CONTAINER BEFOR PALLETIZING
; rung 5
LD 2029.06  ; PALLETIZING CONTAINER
TIM 1814 #1  ; PALLETIZING CONTAINER
; rung 6
LDNOT 2029.06  ; PALLETIZING CONTAINER
TIM 1815 #1  ; NO PALLETIZING CONTAINER
; rung 7
LDNOT 2029.06  ; PALLETIZING CONTAINER
AND 2022.00  ; LOADING CONVEYOR
TIM 1819 #150  ; NO LOADING CONTAINER
; rung 8
LD 2029.07  ; PALLETIZING CONTAINER UPPER SECTION
TIM 1816 #1  ; PALLETIZING CONTAINER UPPER SECTION

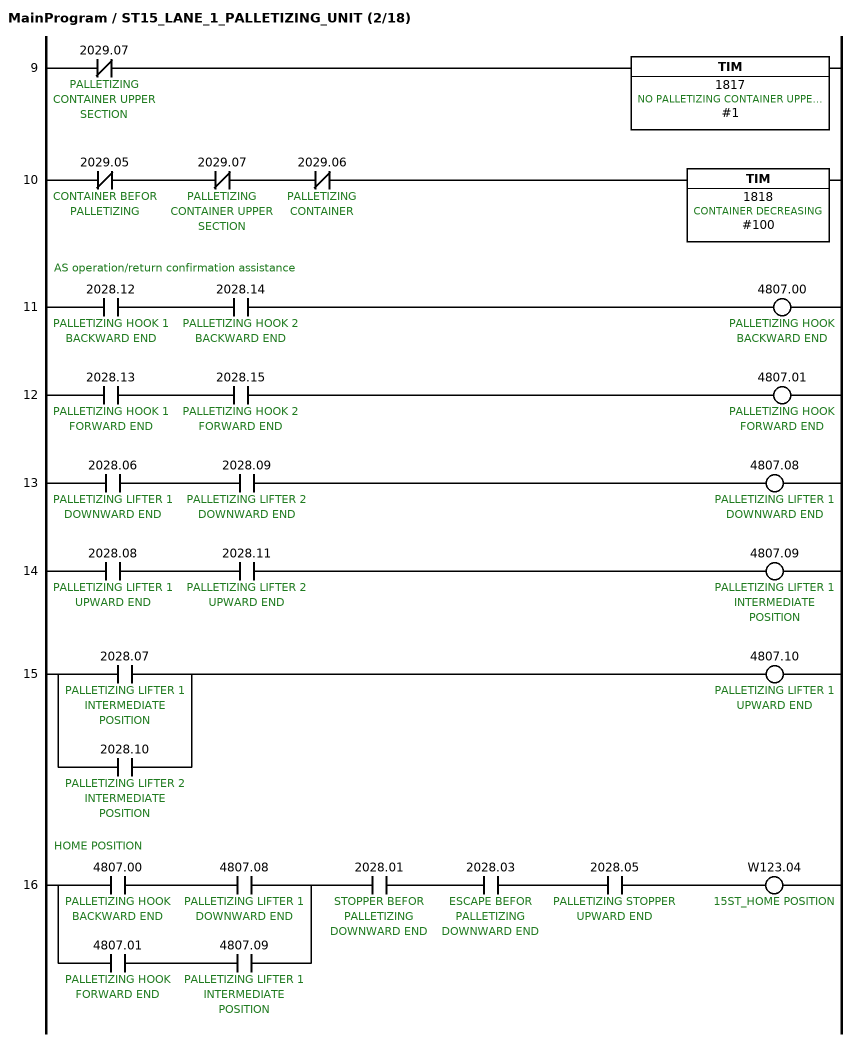
; rung 9
LDNOT 2029.07  ; PALLETIZING CONTAINER UPPER SECTION
TIM 1817 #1  ; NO PALLETIZING CONTAINER UPPER SECTION
; rung 10
LDNOT 2029.05  ; CONTAINER BEFOR PALLETIZING
ANDNOT 2029.07  ; PALLETIZING CONTAINER UPPER SECTION
ANDNOT 2029.06  ; PALLETIZING CONTAINER
TIM 1818 #100  ; CONTAINER DECREASING
; rung 11: AS operation/return confirmation assistance
LD 2028.12  ; PALLETIZING HOOK 1 BACKWARD END
AND 2028.14  ; PALLETIZING HOOK 2 BACKWARD END
OUT 4807.00  ; PALLETIZING HOOK BACKWARD END
; rung 12
LD 2028.13  ; PALLETIZING HOOK 1 FORWARD END
AND 2028.15  ; PALLETIZING HOOK 2 FORWARD END
OUT 4807.01  ; PALLETIZING HOOK FORWARD END
; rung 13
LD 2028.06  ; PALLETIZING LIFTER 1 DOWNWARD END
AND 2028.09  ; PALLETIZING LIFTER 2 DOWNWARD END
OUT 4807.08  ; PALLETIZING LIFTER 1 DOWNWARD END
; rung 14
LD 2028.08  ; PALLETIZING LIFTER 1 UPWARD END
AND 2028.11  ; PALLETIZING LIFTER 2 UPWARD END
OUT 4807.09  ; PALLETIZING LIFTER 1 INTERMEDIATE POSITION
; rung 15
LD 2028.07  ; PALLETIZING LIFTER 1 INTERMEDIATE POSITION
OR 2028.10  ; PALLETIZING LIFTER 2 INTERMEDIATE POSITION
OUT 4807.10  ; PALLETIZING LIFTER 1 UPWARD END
; rung 16: HOME POSITION
LD 4807.00  ; PALLETIZING HOOK BACKWARD END
AND 4807.08  ; PALLETIZING LIFTER 1 DOWNWARD END
LD 4807.01  ; PALLETIZING HOOK FORWARD END
AND 4807.09  ; PALLETIZING LIFTER 1 INTERMEDIATE POSITION
ORLD
AND 2028.01  ; STOPPER BEFOR PALLETIZING DOWNWARD END
AND 2028.03  ; ESCAPE BEFOR PALLETIZING DOWNWARD END
AND 2028.05  ; PALLETIZING STOPPER UPWARD END
OUT W123.04  ; 15ST_HOME POSITION

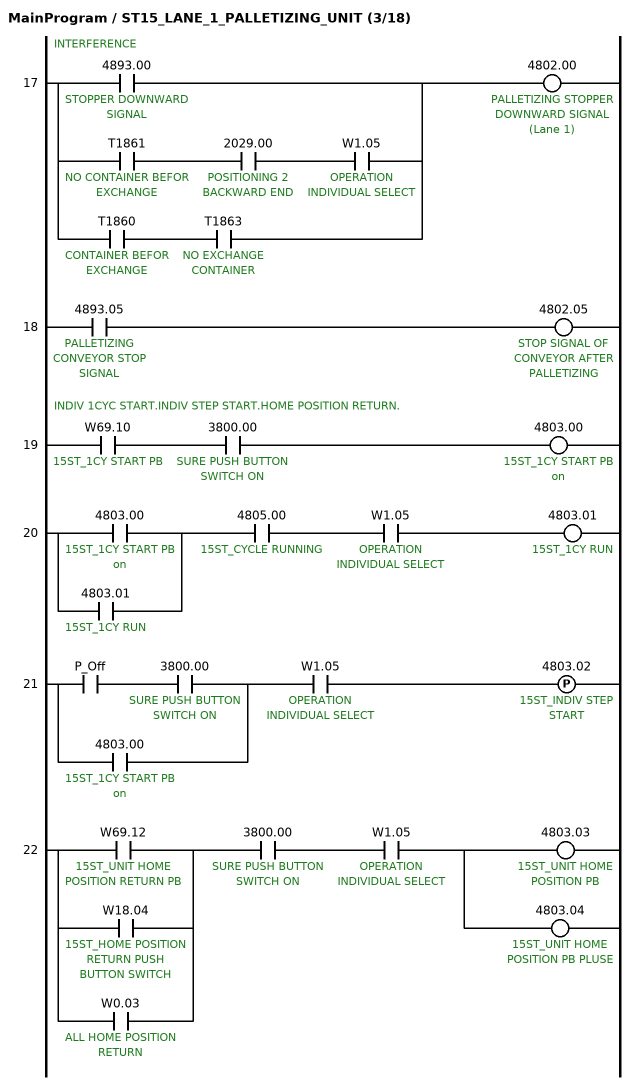
; rung 17: INTERFERENCE
LD 4893.00  ; STOPPER DOWNWARD SIGNAL
LD T1861  ; NO CONTAINER BEFOR EXCHANGE
AND 2029.00  ; POSITIONING 2 BACKWARD END
AND W1.05  ; OPERATION INDIVIDUAL SELECT
ORLD
LD T1860  ; CONTAINER BEFOR EXCHANGE
AND T1863  ; NO EXCHANGE CONTAINER
ORLD
OUT 4802.00  ; PALLETIZING STOPPER DOWNWARD SIGNAL (Lane 1)
; rung 18
LD 4893.05  ; PALLETIZING CONVEYOR STOP SIGNAL
OUT 4802.05  ; STOP SIGNAL OF CONVEYOR AFTER PALLETIZING
; rung 19: INDIV 1CYC START.INDIV STEP START.HOME POSITION RETURN.
LD W69.10  ; 15ST_1CY START PB
AND 3800.00  ; SURE PUSH BUTTON SWITCH ON
OUT 4803.00  ; 15ST_1CY START PB on
; rung 20
LD 4803.00  ; 15ST_1CY START PB on
OR 4803.01  ; 15ST_1CY RUN
AND 4805.00  ; 15ST_CYCLE RUNNING
AND W1.05  ; OPERATION INDIVIDUAL SELECT
OUT 4803.01  ; 15ST_1CY RUN
; rung 21
LD P_Off
AND 3800.00  ; SURE PUSH BUTTON SWITCH ON
OR 4803.00  ; 15ST_1CY START PB on
AND W1.05  ; OPERATION INDIVIDUAL SELECT
DIFU(013) 4803.02  ; 15ST_INDIV STEP START
; rung 22
LD W69.12  ; 15ST_UNIT HOME POSITION RETURN PB
OR W18.04  ; 15ST_HOME POSITION RETURN PUSH BUTTON SWITCH
OR W0.03  ; ALL HOME POSITION RETURN
AND 3800.00  ; SURE PUSH BUTTON SWITCH ON
AND W1.05  ; OPERATION INDIVIDUAL SELECT
OUT 4803.03  ; 15ST_UNIT HOME POSITION PB
OUT 4803.04  ; 15ST_UNIT HOME POSITION PB PLUSE

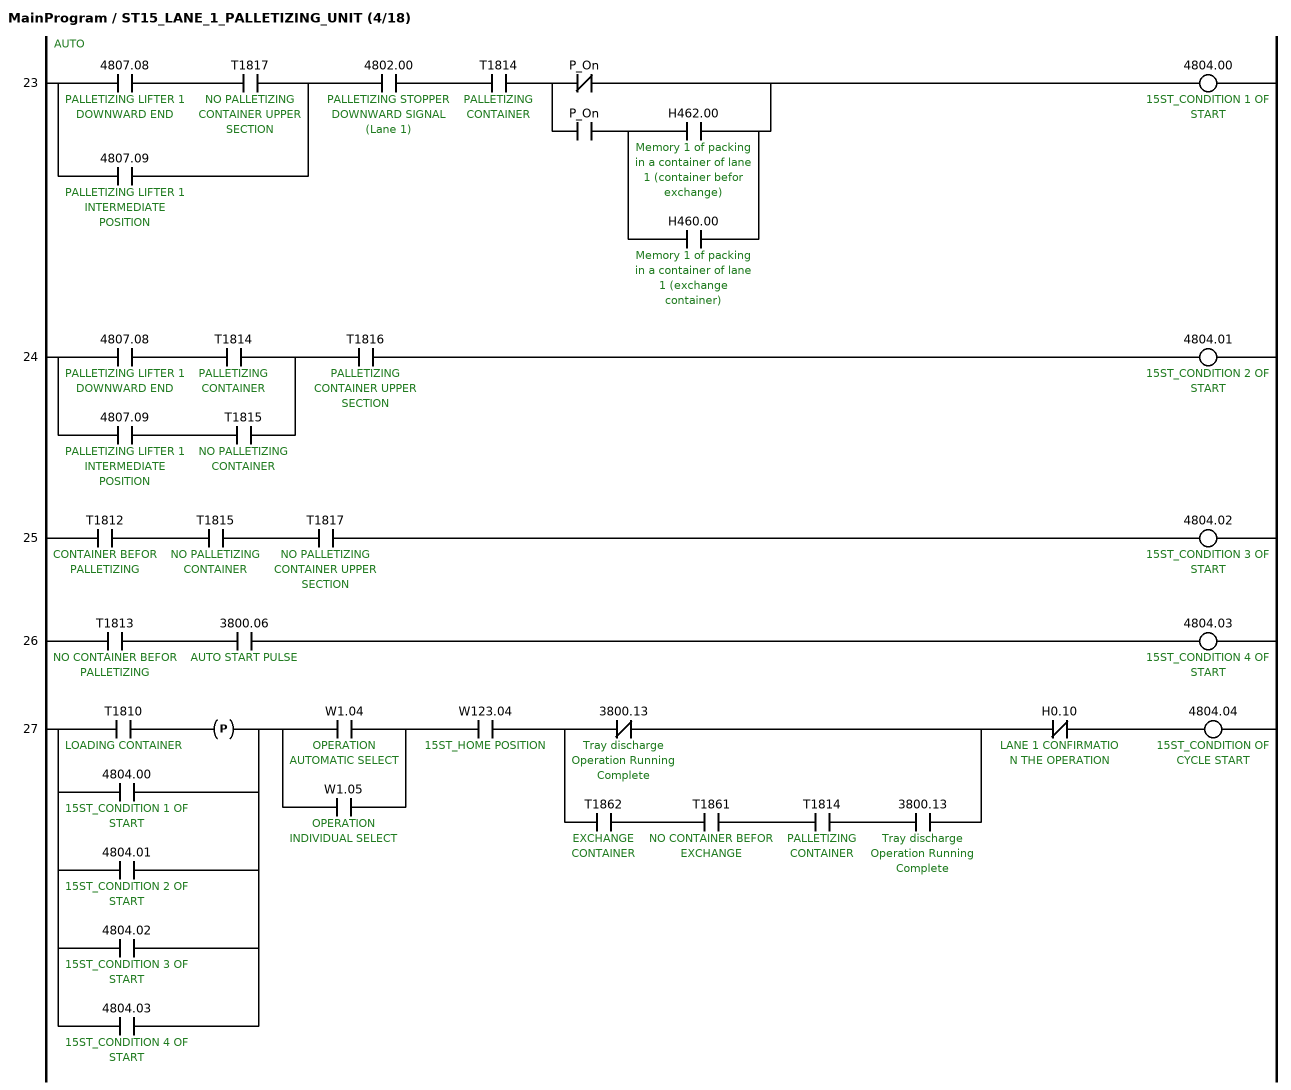
; rung 23: AUTO
LD 4807.08  ; PALLETIZING LIFTER 1 DOWNWARD END
AND T1817  ; NO PALLETIZING CONTAINER UPPER SECTION
OR 4807.09  ; PALLETIZING LIFTER 1 INTERMEDIATE POSITION
AND 4802.00  ; PALLETIZING STOPPER DOWNWARD SIGNAL (Lane 1)
AND T1814  ; PALLETIZING CONTAINER
LDNOT P_On
LD P_On
LD H462.00  ; Memory 1 of packing in a container of lane 1 (container befor exchange)
OR H460.00  ; Memory 1 of packing in a container of lane 1 (exchange container)
ANDLD
ORLD
ANDLD
OUT 4804.00  ; 15ST_CONDITION 1 OF START
; rung 24
LD 4807.08  ; PALLETIZING LIFTER 1 DOWNWARD END
AND T1814  ; PALLETIZING CONTAINER
LD 4807.09  ; PALLETIZING LIFTER 1 INTERMEDIATE POSITION
AND T1815  ; NO PALLETIZING CONTAINER
ORLD
AND T1816  ; PALLETIZING CONTAINER UPPER SECTION
OUT 4804.01  ; 15ST_CONDITION 2 OF START
; rung 25
LD T1812  ; CONTAINER BEFOR PALLETIZING
AND T1815  ; NO PALLETIZING CONTAINER
AND T1817  ; NO PALLETIZING CONTAINER UPPER SECTION
OUT 4804.02  ; 15ST_CONDITION 3 OF START
; rung 26
LD T1813  ; NO CONTAINER BEFOR PALLETIZING
AND 3800.06  ; AUTO START PULSE
OUT 4804.03  ; 15ST_CONDITION 4 OF START
; rung 27
LD T1810  ; LOADING CONTAINER
UP(521)
OR 4804.00  ; 15ST_CONDITION 1 OF START
OR 4804.01  ; 15ST_CONDITION 2 OF START
OR 4804.02  ; 15ST_CONDITION 3 OF START
OR 4804.03  ; 15ST_CONDITION 4 OF START
LD W1.04  ; OPERATION AUTOMATIC SELECT
OR W1.05  ; OPERATION INDIVIDUAL SELECT
ANDLD
AND W123.04  ; 15ST_HOME POSITION
LDNOT 3800.13  ; Tray discharge Operation Running Complete
LD T1862  ; EXCHANGE CONTAINER
AND T1861  ; NO CONTAINER BEFOR EXCHANGE
AND T1814  ; PALLETIZING CONTAINER
AND 3800.13  ; Tray discharge Operation Running Complete
ORLD
ANDLD
ANDNOT H0.10  ; LANE 1 CONFIRMATION THE OPERATION
OUT 4804.04  ; 15ST_CONDITION OF CYCLE START

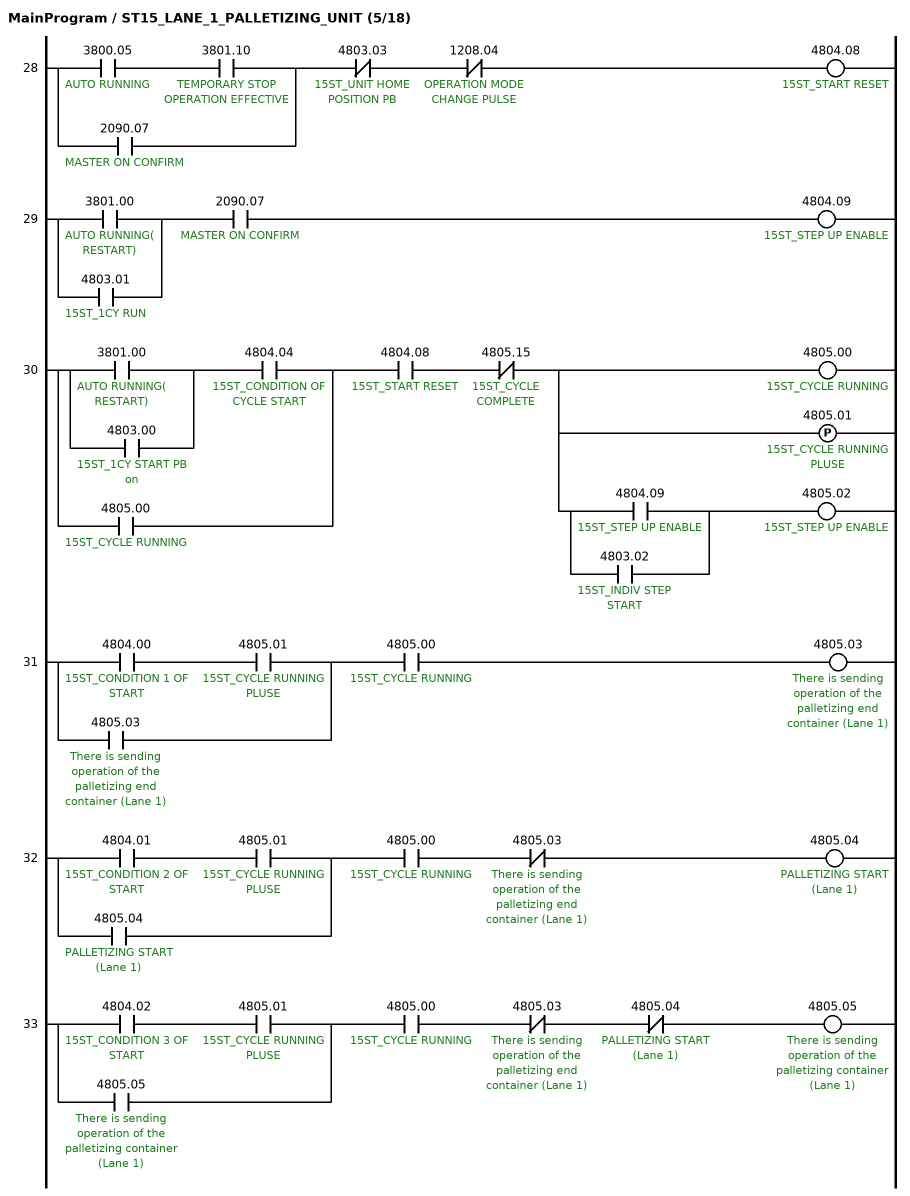
; rung 28
LD 3800.05  ; AUTO RUNNING
AND 3801.10  ; TEMPORARY STOP OPERATION EFFECTIVE
OR 2090.07  ; MASTER ON CONFIRM
ANDNOT 4803.03  ; 15ST_UNIT HOME POSITION PB
ANDNOT 1208.04  ; OPERATION MODE CHANGE PULSE
OUT 4804.08  ; 15ST_START RESET
; rung 29
LD 3801.00  ; AUTO RUNNING(RESTART)
OR 4803.01  ; 15ST_1CY RUN
AND 2090.07  ; MASTER ON CONFIRM
OUT 4804.09  ; 15ST_STEP UP ENABLE
; rung 30
LD 3801.00  ; AUTO RUNNING(RESTART)
OR 4803.00  ; 15ST_1CY START PB on
AND 4804.04  ; 15ST_CONDITION OF CYCLE START
OR 4805.00  ; 15ST_CYCLE RUNNING
AND 4804.08  ; 15ST_START RESET
ANDNOT 4805.15  ; 15ST_CYCLE COMPLETE
OUT 4805.00  ; 15ST_CYCLE RUNNING
DIFU(013) 4805.01  ; 15ST_CYCLE RUNNING PLUSE
LD 4804.09  ; 15ST_STEP UP ENABLE
OR 4803.02  ; 15ST_INDIV STEP START
ANDLD
OUT 4805.02  ; 15ST_STEP UP ENABLE
; rung 31
LD 4804.00  ; 15ST_CONDITION 1 OF START
AND 4805.01  ; 15ST_CYCLE RUNNING PLUSE
OR 4805.03  ; There is sending operation of the palletizing end container (Lane 1)
AND 4805.00  ; 15ST_CYCLE RUNNING
OUT 4805.03  ; There is sending operation of the palletizing end container (Lane 1)
; rung 32
LD 4804.01  ; 15ST_CONDITION 2 OF START
AND 4805.01  ; 15ST_CYCLE RUNNING PLUSE
OR 4805.04  ; PALLETIZING START (Lane 1)
AND 4805.00  ; 15ST_CYCLE RUNNING
ANDNOT 4805.03  ; There is sending operation of the palletizing end container (Lane 1)
OUT 4805.04  ; PALLETIZING START (Lane 1)
; rung 33
LD 4804.02  ; 15ST_CONDITION 3 OF START
AND 4805.01  ; 15ST_CYCLE RUNNING PLUSE
OR 4805.05  ; There is sending operation of the palletizing container (Lane 1)
AND 4805.00  ; 15ST_CYCLE RUNNING
ANDNOT 4805.03  ; There is sending operation of the palletizing end container (Lane 1)
ANDNOT 4805.04  ; PALLETIZING START (Lane 1)
OUT 4805.05  ; There is sending operation of the palletizing container (Lane 1)

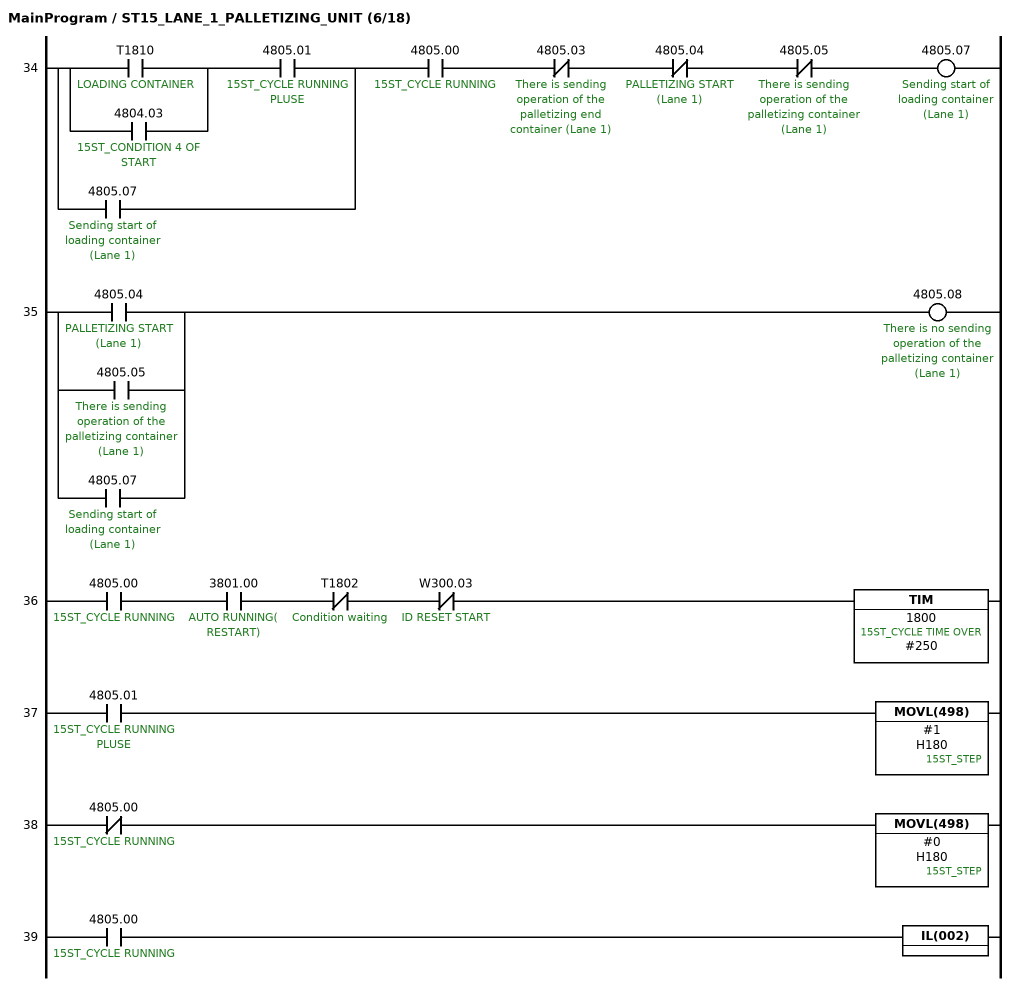
; rung 34
LD T1810  ; LOADING CONTAINER
OR 4804.03  ; 15ST_CONDITION 4 OF START
AND 4805.01  ; 15ST_CYCLE RUNNING PLUSE
OR 4805.07  ; Sending start of loading container (Lane 1)
AND 4805.00  ; 15ST_CYCLE RUNNING
ANDNOT 4805.03  ; There is sending operation of the palletizing end container (Lane 1)
ANDNOT 4805.04  ; PALLETIZING START (Lane 1)
ANDNOT 4805.05  ; There is sending operation of the palletizing container (Lane 1)
OUT 4805.07  ; Sending start of loading container (Lane 1)
; rung 35
LD 4805.04  ; PALLETIZING START (Lane 1)
OR 4805.05  ; There is sending operation of the palletizing container (Lane 1)
OR 4805.07  ; Sending start of loading container (Lane 1)
OUT 4805.08  ; There is no sending operation of the palletizing container (Lane 1)
; rung 36
LD 4805.00  ; 15ST_CYCLE RUNNING
AND 3801.00  ; AUTO RUNNING(RESTART)
ANDNOT T1802  ; Condition waiting
ANDNOT W300.03  ; ID RESET START
TIM 1800 #250  ; 15ST_CYCLE TIME OVER
; rung 37
LD 4805.01  ; 15ST_CYCLE RUNNING PLUSE
MOVL(498) #1 H180  ; 15ST_STEP
; rung 38
LDNOT 4805.00  ; 15ST_CYCLE RUNNING
MOVL(498) #0 H180  ; 15ST_STEP
; rung 39
LD 4805.00  ; 15ST_CYCLE RUNNING
IL(002)

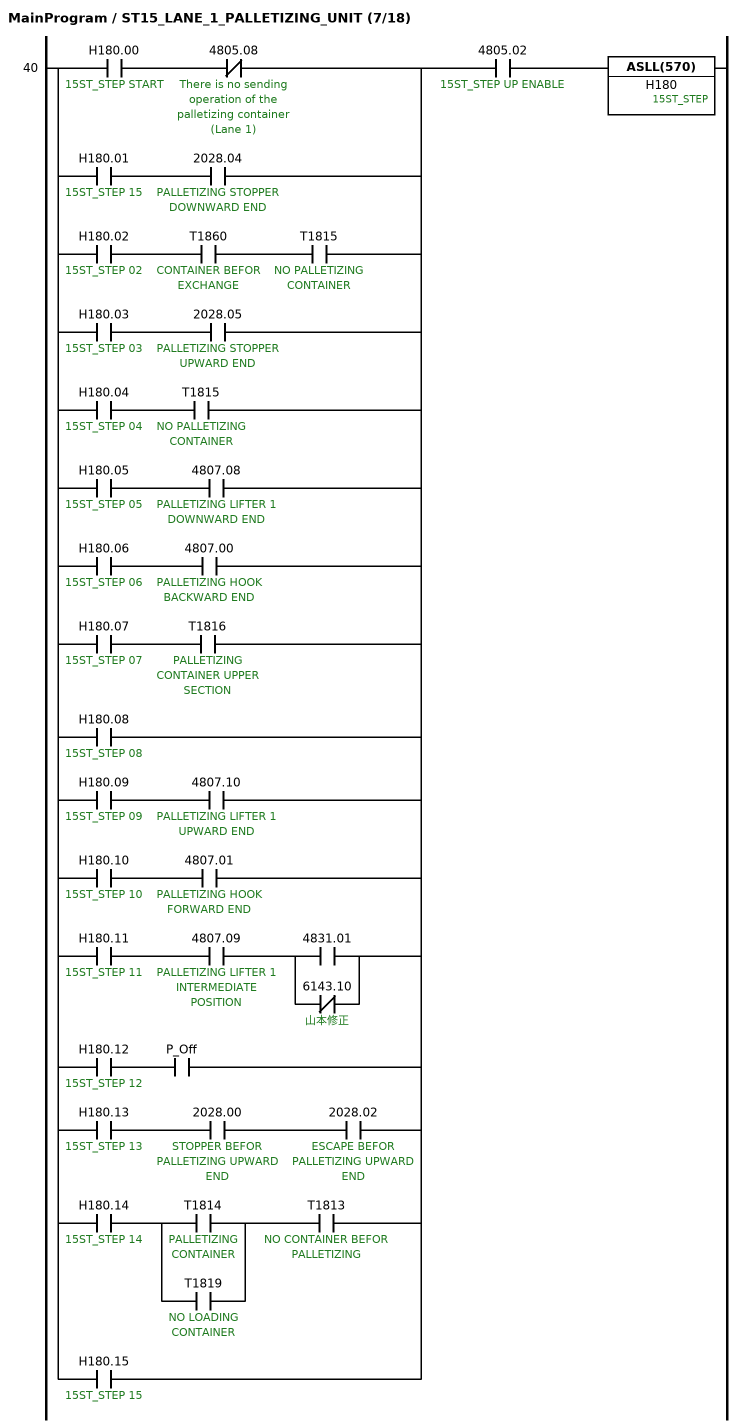
; rung 40
LD H180.00  ; 15ST_STEP START
ANDNOT 4805.08  ; There is no sending operation of the palletizing container (Lane 1)
LD H180.01  ; 15ST_STEP 15
AND 2028.04  ; PALLETIZING STOPPER DOWNWARD END
ORLD
LD H180.02  ; 15ST_STEP 02
AND T1860  ; CONTAINER BEFOR EXCHANGE
AND T1815  ; NO PALLETIZING CONTAINER
ORLD
LD H180.03  ; 15ST_STEP 03
AND 2028.05  ; PALLETIZING STOPPER UPWARD END
ORLD
LD H180.04  ; 15ST_STEP 04
AND T1815  ; NO PALLETIZING CONTAINER
ORLD
LD H180.05  ; 15ST_STEP 05
AND 4807.08  ; PALLETIZING LIFTER 1 DOWNWARD END
ORLD
LD H180.06  ; 15ST_STEP 06
AND 4807.00  ; PALLETIZING HOOK BACKWARD END
ORLD
LD H180.07  ; 15ST_STEP 07
AND T1816  ; PALLETIZING CONTAINER UPPER SECTION
ORLD
OR H180.08  ; 15ST_STEP 08
LD H180.09  ; 15ST_STEP 09
AND 4807.10  ; PALLETIZING LIFTER 1 UPWARD END
ORLD
LD H180.10  ; 15ST_STEP 10
AND 4807.01  ; PALLETIZING HOOK FORWARD END
ORLD
LD H180.11  ; 15ST_STEP 11
AND 4807.09  ; PALLETIZING LIFTER 1 INTERMEDIATE POSITION
LD 4831.01
ORNOT 6143.10  ; 山本修正
ANDLD
ORLD
LD H180.12  ; 15ST_STEP 12
AND P_Off
ORLD
LD H180.13  ; 15ST_STEP 13
AND 2028.00  ; STOPPER BEFOR PALLETIZING UPWARD END
AND 2028.02  ; ESCAPE BEFOR PALLETIZING UPWARD END
ORLD
LD H180.14  ; 15ST_STEP 14
LD T1814  ; PALLETIZING CONTAINER
OR T1819  ; NO LOADING CONTAINER
ANDLD
AND T1813  ; NO CONTAINER BEFOR PALLETIZING
ORLD
OR H180.15  ; 15ST_STEP 15
AND 4805.02  ; 15ST_STEP UP ENABLE
ASLL(570) H180  ; 15ST_STEP

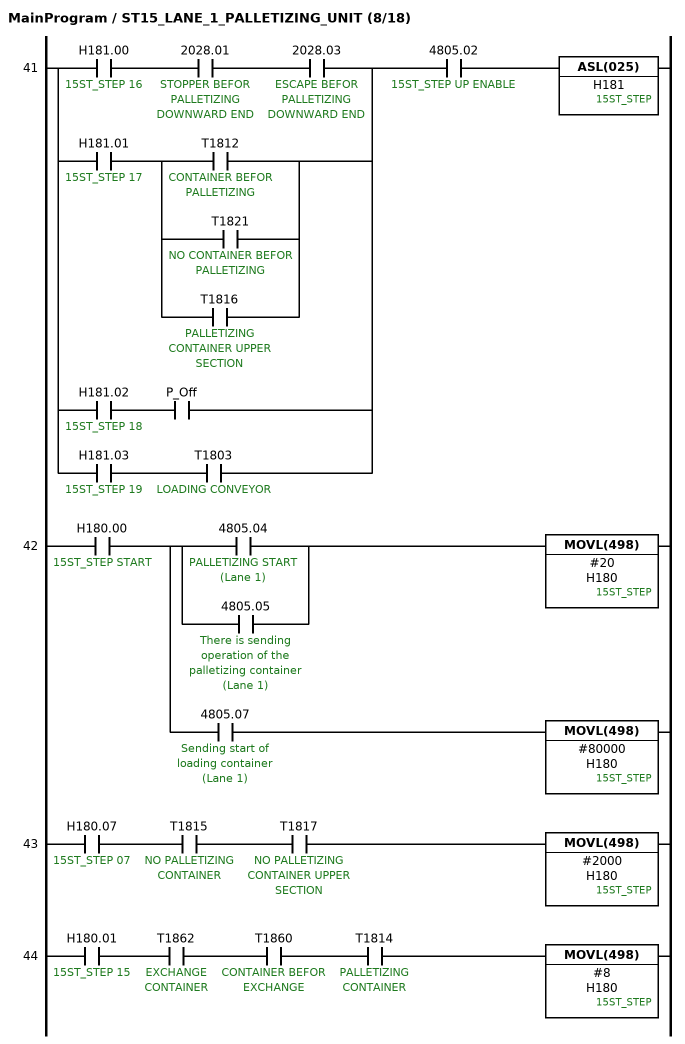
; rung 41
LD H181.00  ; 15ST_STEP 16
AND 2028.01  ; STOPPER BEFOR PALLETIZING DOWNWARD END
AND 2028.03  ; ESCAPE BEFOR PALLETIZING DOWNWARD END
LD H181.01  ; 15ST_STEP 17
LD T1812  ; CONTAINER BEFOR PALLETIZING
OR T1821  ; NO CONTAINER BEFOR PALLETIZING
OR T1816  ; PALLETIZING CONTAINER UPPER SECTION
ANDLD
ORLD
LD H181.02  ; 15ST_STEP 18
AND P_Off
ORLD
LD H181.03  ; 15ST_STEP 19
AND T1803  ; LOADING CONVEYOR
ORLD
AND 4805.02  ; 15ST_STEP UP ENABLE
ASL(025) H181  ; 15ST_STEP
; rung 42
LD H180.00  ; 15ST_STEP START
OUT TR0
LD 4805.04  ; PALLETIZING START (Lane 1)
OR 4805.05  ; There is sending operation of the palletizing container (Lane 1)
ANDLD
MOVL(498) #20 H180  ; 15ST_STEP
LD TR0
AND 4805.07  ; Sending start of loading container (Lane 1)
MOVL(498) #80000 H180  ; 15ST_STEP
; rung 43
LD H180.07  ; 15ST_STEP 07
AND T1815  ; NO PALLETIZING CONTAINER
AND T1817  ; NO PALLETIZING CONTAINER UPPER SECTION
MOVL(498) #2000 H180  ; 15ST_STEP
; rung 44
LD H180.01  ; 15ST_STEP 15
AND T1862  ; EXCHANGE CONTAINER
AND T1860  ; CONTAINER BEFOR EXCHANGE
AND T1814  ; PALLETIZING CONTAINER
MOVL(498) #8 H180  ; 15ST_STEP

